Yaskawa INFORM job: SHESTHREATENINGME.JBI

/JOB
//NAME SHESTHREATENINGME
//POS
///NPOS 2,0,0,0,0,0
///TOOL 0
///POSTYPE PULSE
///PULSE
C00000=2192,31798,-25431,921,-30448,-1591
C00001=2192,20434,-21683,747,-40263,-1449
//INST
///DATE 2026/04/29 01:40
///ATTR SC,RW
///GROUP1 RB1
NOP
MOVJ C00000 VJ=0.78
MOVJ C00001 VJ=0.78
END
